FUNCTION_BLOCK G_10Events_5Unused (* Basic FB with empty ECC *)
  (* Standard: 61499-2 *)
  (* Version 1.0, 2023-09-22, AK124910 *)
  PACKAGE servSeq;
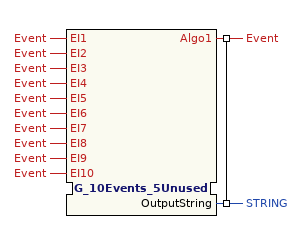
  EVENT_INPUT
    EI1;
    EI2;
    EI3;
    EI4;
    EI5;
    EI6;
    EI7;
    EI8;
    EI9;
    EI10;
  END_EVENT
  EVENT_OUTPUT
    Algo1 WITH OutputString;
  END_EVENT
  VAR_OUTPUT
    OutputString : STRING;
  END_VAR
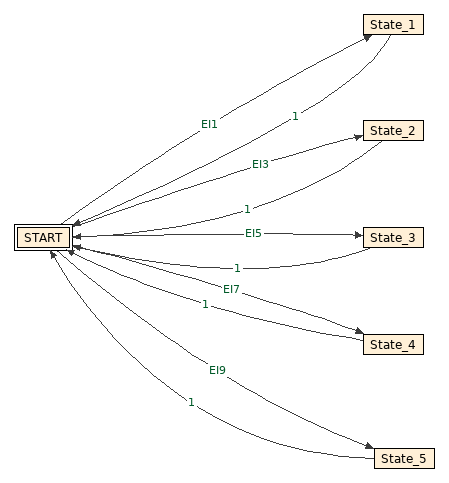
  EC_STATES
    START; (* Initial State *)
    State_1;
    State_2;
    State_3;
    State_4;
    State_5;
  END_STATES
  EC_TRANSITIONS
    START TO State_1 := EI1;
    State_1 TO START := 1;
    START TO State_2 := EI3;
    State_2 TO START := 1;
    START TO State_3 := EI5;
    State_3 TO START := 1;
    START TO State_4 := EI7;
    State_4 TO START := 1;
    START TO State_5 := EI9;
    State_5 TO START := 1;
  END_TRANSITIONS
  (* Service external/internal_interface: Basic FB with empty ECC *)
END_FUNCTION_BLOCK
